FUNCTION TryConvert_LINT_TO_UINT : BOOL
VAR_INPUT
	in : LINT;
	out : REFERENCE TO UINT;
END_VAR

IF in > DatatypeLimits.MAX_VALUE_OF_LINT_WHICH_CAN_BE_HELD_IN_A_UINT THEN
	RETURN;
END_IF

IF in < DatatypeLimits.MIN_VALUE_OF_LINT_WHICH_CAN_BE_HELD_IN_A_UINT THEN
	RETURN;
END_IF

out := LINT_TO_UINT(in);
TryConvert_LINT_TO_UINT := TRUE;

END_FUNCTION

(* stored: Version 1.1.0.1, ProductVersion 3.1.4024.12
   POU TryConvert_LINT_TO_UINT: Id {399484ef-5548-473f-a9df-0e03c1eed061}, SpecialFunc None *)
